INTERFACE I_Mode

METHOD Auto
VAR_INPUT
	bEnable : BOOL;
END_VAR
END_METHOD

METHOD Manual
VAR_INPUT
	bEnable : BOOL;
END_VAR
END_METHOD

METHOD Off
VAR_INPUT
	bEnable : BOOL;
END_VAR
END_METHOD

END_INTERFACE

(* stored: Version 1.1.0.1, ProductVersion 3.1.4024.10
   Itf I_Mode: Id {8cbb066e-df4b-4dc1-bdb7-87eb5200fda7}
   Method Auto: Id {0f9cd9fa-898f-45f9-84b0-e5fe12c05d03}
   Method Manual: Id {cb2e5dfc-81ea-417d-b724-a61cde2b1319}
   Method Off: Id {d23f8b33-20b2-48cc-b0ee-a97946b7d659} *)
